# EPICS substitutions: DMM2kApp/Db/user.substitutions
# Example substitutions file

file "db/dbExample1.db" {
    { user = "kgofron" }
}

file db/dbExample2.db {
    pattern { user, no, scan }
        { "kgofron", 1, "1 second" }
        { "kgofron", 2, "2 second" }
        { "kgofron", 3, "5 second" }
}
